% RSLogix 500 project THREE-PHASE MOTOR CONTROL F-R JOG 3PSS DIR CHNG.RSS, saved by version 10.00.00.00 %
PROJECT "MRLEIGH"    % processor: Bul.1763 MicroLogix 1100 Series B %

PROGRAM FILES
  LAD 2 "MAIN"  16 rungs  % Invert Signals Wired Failsafe %

DATA FILES
  O0 OUTPUT  4 elements
  I1 INPUT  6 elements
  S2 STATUS  66 elements
  B3 BINARY  1 elements
  T4 TIMER  1 elements
  C5 COUNTER  1 elements
  R6 CONTROL  1 elements
  N7 INTEGER  1 elements
  F8 FLOAT  1 elements

LADDER 2 "MAIN"    % Invert Signals Wired Failsafe %
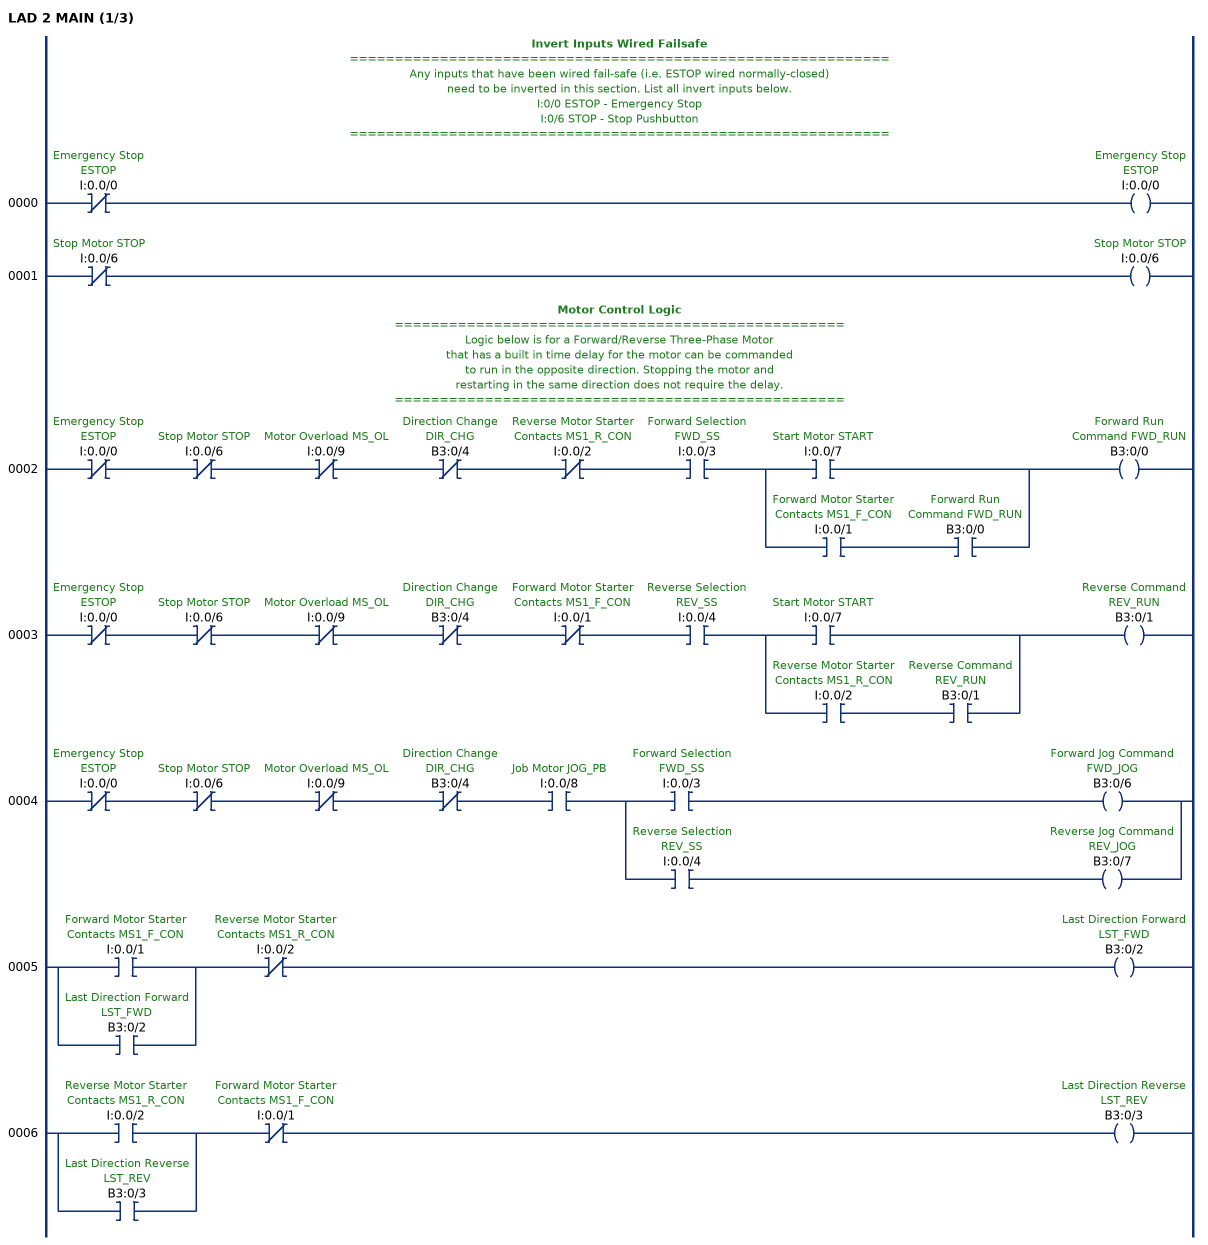
% Rung: 0 %
% TITLE: Invert Inputs Wired Failsafe %
% ============================================================
% 
%   Any inputs that have been wired fail-safe (i.e. ESTOP wired normally-closed)
%   need to be inverted in this section. List all invert inputs below.
% 
%      I:0/0 ESTOP - Emergency Stop
%      I:0/6 STOP - Stop Pushbutton
% 
% ============================================================ %
SOR XIO I:0.0/0 OTE I:0.0/0 EOR
%   I:0.0/0  ESTOP  "Emergency Stop" %
% Rung: 1 %
SOR XIO I:0.0/6 OTE I:0.0/6 EOR
%   I:0.0/6  STOP  "Stop Motor" %
% Rung: 2 %
% TITLE: Motor Control Logic %
% ==================================================
% 
%  Logic below is for a Forward/Reverse Three-Phase Motor
%  that has a built in time delay for the motor can be commanded
%  to run in the opposite direction. Stopping the motor and
%  restarting in the same direction does not require the delay.
% 
% ================================================== %
SOR XIO I:0.0/0 XIO I:0.0/6 XIO I:0.0/9 XIO B3:0/4 XIO I:0.0/2 XIC I:0.0/3 BST XIC I:0.0/7 NXB XIC I:0.0/1 XIC B3:0/0 BND OTE B3:0/0 EOR
%   I:0.0/0  ESTOP  "Emergency Stop" %
%   I:0.0/6  STOP  "Stop Motor" %
%   I:0.0/9  MS_OL  "Motor Overload" %
%   B3:0/4  DIR_CHG  "Direction Change" %
%   I:0.0/2  MS1_R_CON  "Reverse Motor Starter Contacts" %
%   I:0.0/3  FWD_SS  "Forward Selection" %
%   I:0.0/7  START  "Start Motor" %
%   I:0.0/1  MS1_F_CON  "Forward Motor Starter Contacts" %
%   B3:0/0  FWD_RUN  "Forward Run Command" %
% Rung: 3 %
SOR XIO I:0.0/0 XIO I:0.0/6 XIO I:0.0/9 XIO B3:0/4 XIO I:0.0/1 XIC I:0.0/4 BST XIC I:0.0/7 NXB XIC I:0.0/2 XIC B3:0/1 BND OTE B3:0/1 EOR
%   I:0.0/0  ESTOP  "Emergency Stop" %
%   I:0.0/6  STOP  "Stop Motor" %
%   I:0.0/9  MS_OL  "Motor Overload" %
%   B3:0/4  DIR_CHG  "Direction Change" %
%   I:0.0/1  MS1_F_CON  "Forward Motor Starter Contacts" %
%   I:0.0/4  REV_SS  "Reverse Selection" %
%   I:0.0/7  START  "Start Motor" %
%   I:0.0/2  MS1_R_CON  "Reverse Motor Starter Contacts" %
%   B3:0/1  REV_RUN  "Reverse Command" %
% Rung: 4 %
SOR XIO I:0.0/0 XIO I:0.0/6 XIO I:0.0/9 XIO B3:0/4 XIC I:0.0/8 BST XIC I:0.0/3 OTE B3:0/6 NXB XIC I:0.0/4 OTE B3:0/7 BND EOR
%   I:0.0/0  ESTOP  "Emergency Stop" %
%   I:0.0/6  STOP  "Stop Motor" %
%   I:0.0/9  MS_OL  "Motor Overload" %
%   B3:0/4  DIR_CHG  "Direction Change" %
%   I:0.0/8  JOG_PB  "Job Motor" %
%   I:0.0/3  FWD_SS  "Forward Selection" %
%   B3:0/6  FWD_JOG  "Forward Jog Command" %
%   I:0.0/4  REV_SS  "Reverse Selection" %
%   B3:0/7  REV_JOG  "Reverse Jog Command" %
% Rung: 5 %
SOR BST XIC I:0.0/1 NXB XIC B3:0/2 BND XIO I:0.0/2 OTE B3:0/2 EOR
%   I:0.0/1  MS1_F_CON  "Forward Motor Starter Contacts" %
%   B3:0/2  LST_FWD  "Last Direction Forward" %
%   I:0.0/2  MS1_R_CON  "Reverse Motor Starter Contacts" %
% Rung: 6 %
SOR BST XIC I:0.0/2 NXB XIC B3:0/3 BND XIO I:0.0/1 OTE B3:0/3 EOR
%   I:0.0/2  MS1_R_CON  "Reverse Motor Starter Contacts" %
%   B3:0/3  LST_REV  "Last Direction Reverse" %
%   I:0.0/1  MS1_F_CON  "Forward Motor Starter Contacts" %

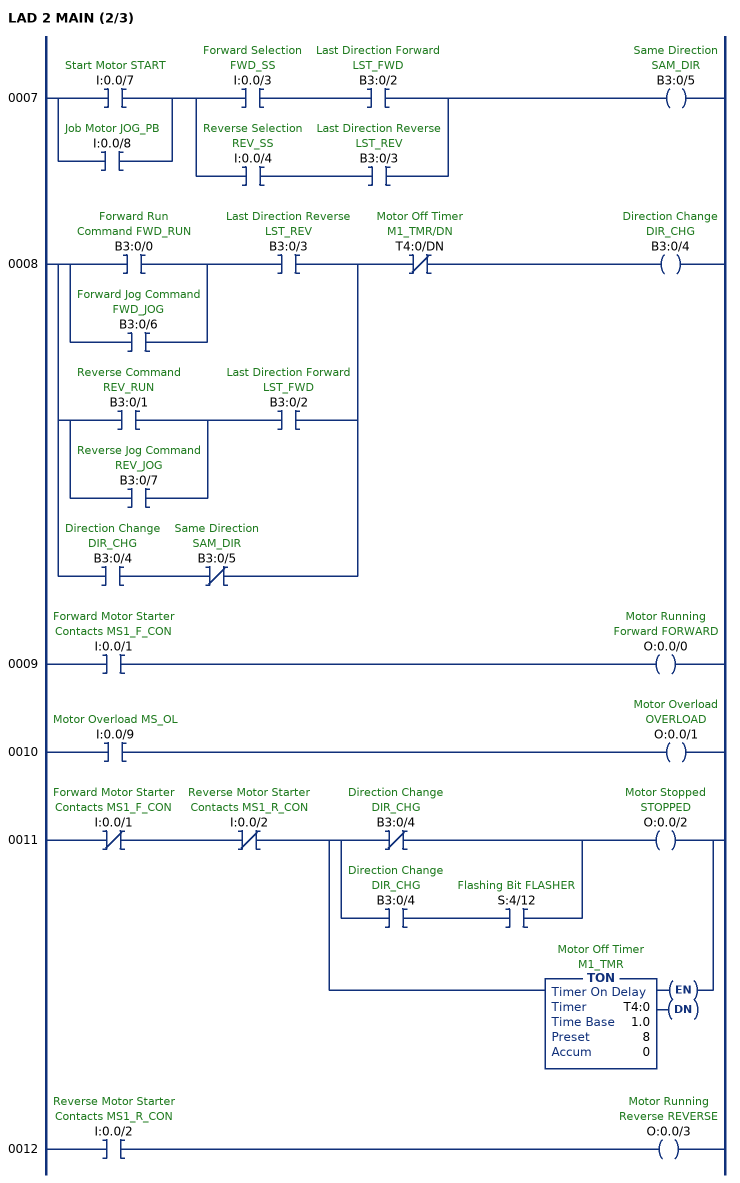
% Rung: 7 %
SOR BST XIC I:0.0/7 NXB XIC I:0.0/8 BND BST XIC I:0.0/3 XIC B3:0/2 NXB XIC I:0.0/4 XIC B3:0/3 BND OTE B3:0/5 EOR
%   I:0.0/7  START  "Start Motor" %
%   I:0.0/8  JOG_PB  "Job Motor" %
%   I:0.0/3  FWD_SS  "Forward Selection" %
%   B3:0/2  LST_FWD  "Last Direction Forward" %
%   I:0.0/4  REV_SS  "Reverse Selection" %
%   B3:0/3  LST_REV  "Last Direction Reverse" %
%   B3:0/5  SAM_DIR  "Same Direction" %
% Rung: 8 %
SOR BST BST XIC B3:0/0 NXB XIC B3:0/6 BND XIC B3:0/3 NXB BST XIC B3:0/1 NXB XIC B3:0/7 BND XIC B3:0/2 NXB XIC B3:0/4 XIO B3:0/5 BND XIO T4:0/DN OTE B3:0/4 EOR
%   B3:0/0  FWD_RUN  "Forward Run Command" %
%   B3:0/6  FWD_JOG  "Forward Jog Command" %
%   B3:0/3  LST_REV  "Last Direction Reverse" %
%   B3:0/1  REV_RUN  "Reverse Command" %
%   B3:0/7  REV_JOG  "Reverse Jog Command" %
%   B3:0/2  LST_FWD  "Last Direction Forward" %
%   B3:0/4  DIR_CHG  "Direction Change" %
%   B3:0/5  SAM_DIR  "Same Direction" %
%   T4:0  M1_TMR  "Motor Off Timer" %
% Rung: 9 %
SOR XIC I:0.0/1 OTE O:0.0/0 EOR
%   I:0.0/1  MS1_F_CON  "Forward Motor Starter Contacts" %
%   O:0.0/0  FORWARD  "Motor Running Forward" %
% Rung: 10 %
SOR XIC I:0.0/9 OTE O:0.0/1 EOR
%   I:0.0/9  MS_OL  "Motor Overload" %
%   O:0.0/1  OVERLOAD  "Motor Overload" %
% Rung: 11 %
SOR XIO I:0.0/1 XIO I:0.0/2 BST BST XIO B3:0/4 NXB XIC B3:0/4 XIC S:4/12 BND OTE O:0.0/2 NXB TON T4:0 1.0 8 0 BND EOR
%   I:0.0/1  MS1_F_CON  "Forward Motor Starter Contacts" %
%   I:0.0/2  MS1_R_CON  "Reverse Motor Starter Contacts" %
%   B3:0/4  DIR_CHG  "Direction Change" %
%   S:4/12  FLASHER  "Flashing Bit" %
%   O:0.0/2  STOPPED  "Motor Stopped" %
%   T4:0  M1_TMR  "Motor Off Timer" %
% Rung: 12 %
SOR XIC I:0.0/2 OTE O:0.0/3 EOR
%   I:0.0/2  MS1_R_CON  "Reverse Motor Starter Contacts" %
%   O:0.0/3  REVERSE  "Motor Running Reverse" %

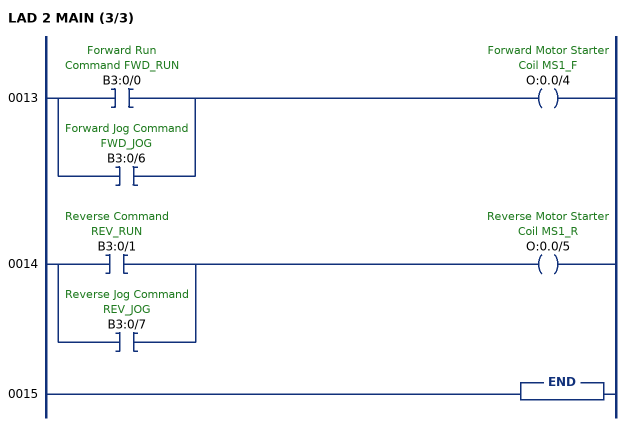
% Rung: 13 %
SOR BST XIC B3:0/0 NXB XIC B3:0/6 BND OTE O:0.0/4 EOR
%   B3:0/0  FWD_RUN  "Forward Run Command" %
%   B3:0/6  FWD_JOG  "Forward Jog Command" %
%   O:0.0/4  MS1_F  "Forward Motor Starter Coil" %
% Rung: 14 %
SOR BST XIC B3:0/1 NXB XIC B3:0/7 BND OTE O:0.0/5 EOR
%   B3:0/1  REV_RUN  "Reverse Command" %
%   B3:0/7  REV_JOG  "Reverse Jog Command" %
%   O:0.0/5  MS1_R  "Reverse Motor Starter Coil" %
% Rung: 15 %
SOR END EOR

OTHER DOCUMENTED ADDRESSES
  PFILE:3  "Simulation"
  PFILE:4  "Main Program"
  U:3  SIM  "Simulation Program File"
  U:4  MAIN  "Main Program File"

DATA TABLE (non-zero values as saved)
DATA B3
% B3:0 % 0X000A
DATA T4
% .PRE .ACC %
% T4:0 % 8 0
